FUNCTION_BLOCK Product_Recipe (* Basic Function Block Type *)
  (* Standard: 61499-2 *)
  (* Version 0.0, 4/22/2020, prana, nxtControl GmbH, Template *)
  PACKAGE Main;
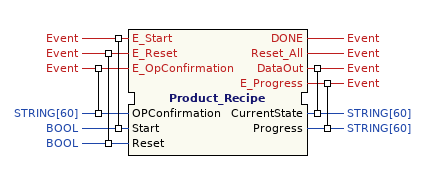
  EVENT_INPUT
    E_Start WITH Start; (* Initialization Request *) {SET_ATTRIBUTE(Runtime.OPCUA.Access, 2)}
    E_Reset WITH Reset;
    E_OpConfirmation WITH OPConfirmation;
  END_EVENT
  EVENT_OUTPUT
    DONE;
    Reset_All;
    DataOut WITH CurrentState;
    E_Progress WITH Progress;
  END_EVENT
  VAR_INPUT
    OPConfirmation : STRING[60];
    Start : BOOL;
    Reset : BOOL;
  END_VAR
  VAR_OUTPUT
    CurrentState : STRING[60];
    Progress : STRING[60];
  END_VAR
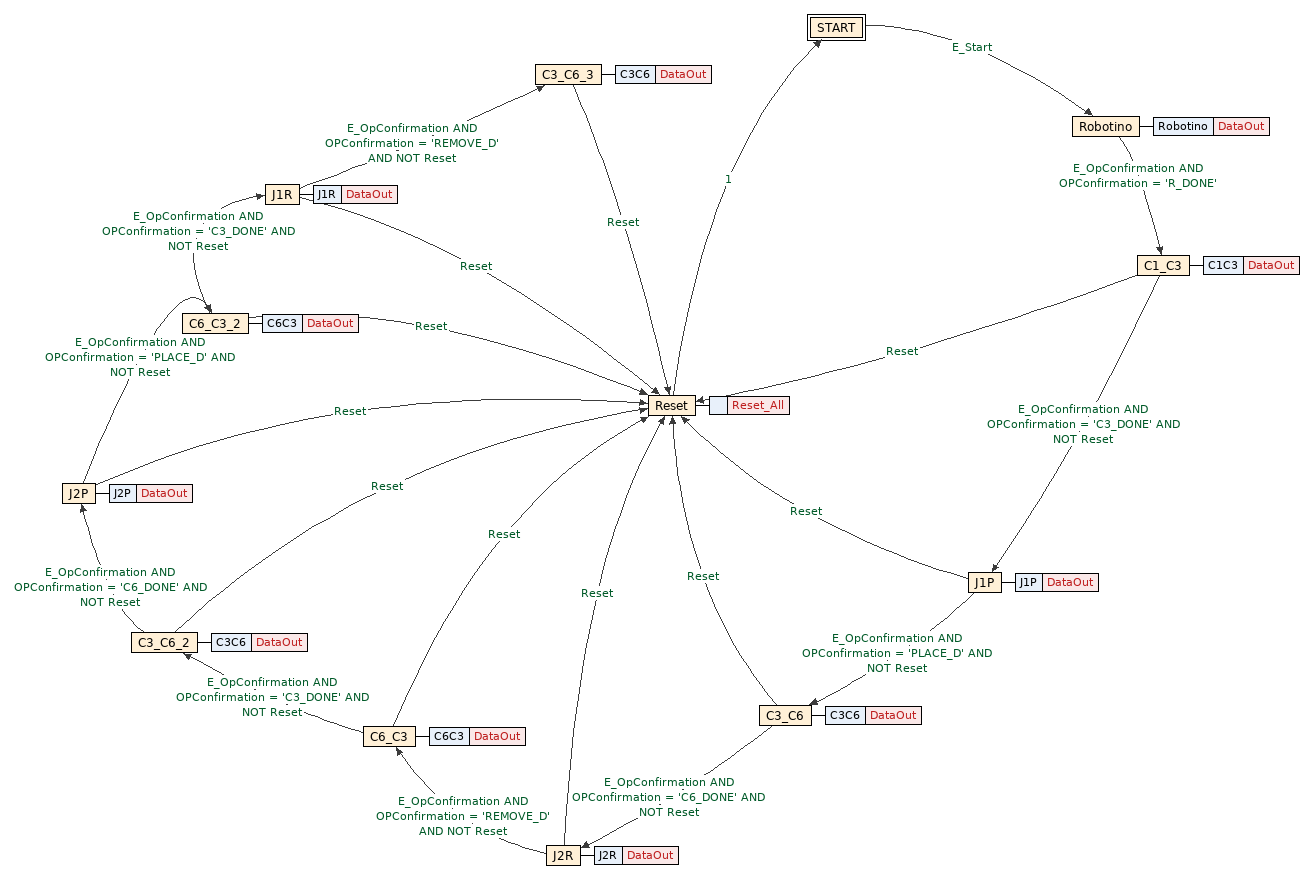
  EC_STATES
    START; (* Initial State *)
    Robotino : Robotino -> DataOut;
    J1P : J1P -> DataOut;
    C3_C6 : C3C6 -> DataOut;
    C1_C3 : C1C3 -> DataOut;
    J2R : J2R -> DataOut;
    C6_C3 : C6C3 -> DataOut;
    C3_C6_2 : C3C6 -> DataOut;
    J2P : J2P -> DataOut;
    C6_C3_2 : C6C3 -> DataOut;
    J1R : J1R -> DataOut;
    C3_C6_3 : C3C6 -> DataOut;
    Reset : -> Reset_All;
  END_STATES
  EC_TRANSITIONS
    START TO Robotino := E_Start;
    J1P TO C3_C6 := E_OpConfirmation AND OPConfirmation = 'PLACE_D' AND NOT Reset;
    Robotino TO C1_C3 := E_OpConfirmation AND OPConfirmation = 'R_DONE';
    C3_C6 TO J2R := E_OpConfirmation AND OPConfirmation = 'C6_DONE' AND NOT Reset;
    J2R TO C6_C3 := E_OpConfirmation AND OPConfirmation = 'REMOVE_D' AND NOT Reset;
    C6_C3 TO C3_C6_2 := E_OpConfirmation AND OPConfirmation = 'C3_DONE' AND NOT Reset;
    C3_C6_2 TO J2P := E_OpConfirmation AND OPConfirmation = 'C6_DONE' AND NOT Reset;
    J2P TO C6_C3_2 := E_OpConfirmation AND OPConfirmation = 'PLACE_D' AND NOT Reset;
    C6_C3_2 TO J1R := E_OpConfirmation AND OPConfirmation = 'C3_DONE' AND NOT Reset;
    J1R TO C3_C6_3 := E_OpConfirmation AND OPConfirmation = 'REMOVE_D' AND NOT Reset;
    C1_C3 TO J1P := E_OpConfirmation AND OPConfirmation = 'C3_DONE' AND NOT Reset;
    C3_C6_2 TO Reset := Reset;
    C6_C3 TO Reset := Reset;
    J2P TO Reset := Reset;
    C6_C3_2 TO Reset := Reset;
    J1R TO Reset := Reset;
    C3_C6_3 TO Reset := Reset;
    J2R TO Reset := Reset;
    C3_C6 TO Reset := Reset;
    J1P TO Reset := Reset;
    C1_C3 TO Reset := Reset;
    Reset TO START := 1;
  END_TRANSITIONS
  ALGORITHM Robotino IN ST:
CurrentState :='R_START';
  END_ALGORITHM
  ALGORITHM C1_C2 IN ST:
CurrentState := 'C1_to_C2';
  END_ALGORITHM
  ALGORITHM J1P IN ST:
CurrentState := 'J1P';
  END_ALGORITHM
  ALGORITHM C2C3 IN ST:
CurrentState := 'C2_to_C3';
  END_ALGORITHM
  ALGORITHM C3C6 IN ST:
CurrentState := 'C3_to_C6';
  END_ALGORITHM
  ALGORITHM C6C3 IN ST:
CurrentState := 'C6_to_C3';
  END_ALGORITHM
  ALGORITHM J1R IN ST:
CurrentState := 'J1R';
  END_ALGORITHM
  ALGORITHM J2P IN ST:
CurrentState := 'J2P';
  END_ALGORITHM
  ALGORITHM C6C4 IN ST:
CurrentState := 'C6_to_C4';
  END_ALGORITHM
  ALGORITHM C4_C6 IN ST:
CurrentState := 'C4_to_C6';
  END_ALGORITHM
  ALGORITHM J2R IN ST:
CurrentState := 'J2R';
  END_ALGORITHM
  ALGORITHM C1C3 IN ST:
CurrentState := 'C1_to_C3';
  END_ALGORITHM
END_FUNCTION_BLOCK
